SUBAPPLICATION tastend (* Subapplication Type *)
  (* Standard: 61499-2 *)
  (* Version 1.0, 2024-10-23, franz *)
  PACKAGE FBs::Uebungen::Uebung_103::subapp;
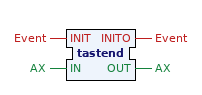
  EVENT_INPUT
    INIT; (* Initialization Request *)
  END_EVENT
  EVENT_OUTPUT
    INITO; (* Initialization Confirm *)
  END_EVENT
  SOCKETS
    IN : AX;
  END_SOCKETS
  PLUGS
    OUT : AX;
  END_PLUGS
  EVENT_CONNECTIONS
    INIT TO INITO;
  END_CONNECTIONS
  ADAPTER_CONNECTIONS
    IN TO OUT;
  END_CONNECTIONS
END_SUBAPPLICATION
